INTERFACE I_CanReleaseWhenDone

METHOD PUBLIC ThenRelease
VAR_INPUT
END_VAR
END_METHOD

END_INTERFACE

(* stored: Version 1.1.0.1, ProductVersion 3.1.4024.12
   Itf I_CanReleaseWhenDone: Id {97435b89-20a9-4fae-b395-a48ce0a49a9d}
   Method ThenRelease: Id {19d335de-3bd0-4086-9556-09b2e8260417} *)
